PROGRAM PRG_TCPIP 
VAR	
	bInit 						:BOOL := TRUE;
	
	fbReadFromCameraTCP			:FB_ReadTCP;
	bConnectToReadSocket		:BOOL;
	
	fbWriteToHLZ				:FB_WriteTCP;
	bConnectToWriteSocket		:BOOL;
END_VAR

//Init
IF bInit THEN	
	bInit := FALSE;
END_IF

//Call Methods
M_ReadCameraTCP();
M_WriteToHlzTCP();

METHOD PUBLIC M_ReadCameraTCP : BOOL
VAR_INPUT
END_VAR
VAR
	stTCPConnection				:ST_TCPConnection;
END_VAR
//Initialize Read TCP
stTCPConnection.sRemoteHost := '10.12.5.10';
stTCPConnection.nRemotePort := 51236;
stTCPConnection.tTimeOut := T#45S;
stTCPConnection.bSocketConnect := bConnectToReadSocket;
stTCPConnection.bReset := GVL_ItemSimulator.bResetRegistry;


//Call Read TCP
fbReadFromCameraTCP(stTCPConnection:=stTCPConnection);
END_METHOD

METHOD PUBLIC M_WriteToHlzTCP : BOOL
VAR_INPUT
END_VAR
VAR
	stTCPConnection				:ST_TCPConnection;
END_VAR
//Initialize Write TCP
stTCPConnection.sRemoteHost := '10.12.5.10';
stTCPConnection.nRemotePort := 51236;
stTCPConnection.tTimeOut := T#45S;
stTCPConnection.bSocketConnect := bConnectToWriteSocket;
stTCPConnection.bReset := GVL_ItemSimulator.bResetRegistry;


//Call Write TCP
fbWriteToHLZ(stTCPConnection:=stTCPConnection);
END_METHOD

END_PROGRAM

(* stored: Version 1.1.0.1, ProductVersion 3.1.4024.12
   POU PRG_TCPIP: Id {e26f0609-c5dd-4c0e-bab1-8c4ef3547268}, SpecialFunc None
   Method M_ReadCameraTCP: Id {c95fd805-970b-4ceb-80e0-471b56be01fb}
   Method M_WriteToHlzTCP: Id {b613047a-ae2a-4d62-a218-edbd1edcce5b} *)
